FUNCTION_BLOCK FB_EventLoggerCore EXTENDS TcLogCore

END_FUNCTION_BLOCK

(* stored: Version 1.1.0.1, ProductVersion 3.1.4024.12
   POU FB_EventLoggerCore: Id {0877040a-dfa8-423e-9d31-5def1eafc26d}, SpecialFunc None *)
